{attribute 'qualified_only'}
{attribute 'hide'}
VAR_GLOBAL INTERNAL CONSTANT
  BrakeEpsilon : LREAL := 2.2E-14;
  DoubleEpsilon : LREAL := 2.2204460492503131E-016; // smallest such that 1.0+Constants.DoubleEpsilon != 1.0
  Epsilon : LREAL := 1E-8;
  Epsilon16 : LREAL := 16 * 2.2204460492503131E-016;
  EpsilonColinear : LREAL := 1E-7;
  Infinity : LREAL := 1.7976931348623157E+308;  
  Tolerance : LREAL := 1E-14;
  Cos120 : LREAL := -0.50;
  Sin120 : LREAL := 0.866025403784438646764;  
  Pi : LREAL := 3.14159265358979323846;
  Minimum : LREAL := 1.17549435082E-38;  // used for validating input
  
  VelocityEpsilon : LREAL := 1E-12;
  AccelerationEpsilon : LREAL := 1E-12;
  JerkEpsilon : LREAL := 1E-12; 
  
  PositionPrecision : LREAL := 1E-8;
  VelocityPrecision : LREAL := 1E-8;
  AccelerationPrecision : LREAL := 1E-10;
  TimePrecision : LREAL := 1E-12;  
  
  Tmax : LREAL := 1E12;
END_VAR

(* stored: Version 1.1.0.1
   GVL Constants: Id {2aa9bca8-7d9a-4e76-bf88-1bddc5102572} *)
